Staubli VAL3: writeCFG.pgx

program writeCFG()
  local bool l_bResult
  local num l_nError
  local num l_nItem
  local string l_sValue
begin
  l_nItem=0
  // Update Tool value with data entered by user
  resize(sCaption,1,pg:nNumOfTxtBox)
  call pg:getCaption(sCaption)
  //X
  call pg:getFieldValue(sCaption[l_nItem],l_sValue,l_nError)
  toNum(l_sValue,cfg:tPointer.trsf.x,l_bResult)
  l_nItem=l_nItem+1
  //Y
  call pg:getFieldValue(sCaption[l_nItem],l_sValue,l_nError)
  toNum(l_sValue,cfg:tPointer.trsf.y,l_bResult)
  l_nItem=l_nItem+1
  //Z
  call pg:getFieldValue(sCaption[l_nItem],l_sValue,l_nError)
  toNum(l_sValue,cfg:tPointer.trsf.z,l_bResult)
  l_nItem=l_nItem+1
  //RX
  call pg:getFieldValue(sCaption[l_nItem],l_sValue,l_nError)
  toNum(l_sValue,cfg:tPointer.trsf.rx,l_bResult)
  l_nItem=l_nItem+1
  //RY
  call pg:getFieldValue(sCaption[l_nItem],l_sValue,l_nError)
  toNum(l_sValue,cfg:tPointer.trsf.ry,l_bResult)
  l_nItem=l_nItem+1
  //RZ
  call pg:getFieldValue(sCaption[l_nItem],l_sValue,l_nError)
  toNum(l_sValue,cfg:tPointer.trsf.rz,l_bResult)
  l_nItem=l_nItem+1
  // Approach TRSF
  // X value
  call pg:getFieldValue(sCaption[l_nItem],l_sValue,l_nError)
  toNum(l_sValue,cfg:trApproach.x,l_bResult)
  l_nItem=l_nItem+1
  // Y value
  call pg:getFieldValue(sCaption[l_nItem],l_sValue,l_nError)
  toNum(l_sValue,cfg:trApproach.y,l_bResult)
  l_nItem=l_nItem+1
  // Z value
  call pg:getFieldValue(sCaption[l_nItem],l_sValue,l_nError)
  toNum(l_sValue,cfg:trApproach.z,l_bResult)
  l_nItem=l_nItem+1
  // Enable event logging
  call pg:getFieldValue(sCaption[l_nItem],l_sValue,l_nError)
  toNum(l_sValue,cfg:nLog,l_bResult)
end
